FUNCTION_BLOCK E_CTU (* Event-Driven Up Counter *)
  (* Standard: 61499-1-A.18; Classification: Event-driven blocks; Function: Up-counter *)
  (* Version 0.1, 2001-04-27, JHC, Rockwell Automation, XML version *)
  (* Version 0.0, 1999-01-22, JHC, Rockwell Automation, SRC version *)
  (* Compiler header: package fb.rt.event; *)
  (* Compiler Java IBM VisualAge 3.0 *)
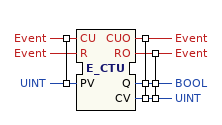
  EVENT_INPUT
    CU WITH PV; (* Count Up *)
    R; (* Reset *)
  END_EVENT
  EVENT_OUTPUT
    CUO WITH Q, CV; (* Count Up Output Event *)
    RO WITH Q, CV; (* Reset Output Event *)
  END_EVENT
  VAR_INPUT
    PV : UINT; (* Preset Value *)
  END_VAR
  VAR_OUTPUT
    Q : BOOL; (* CV==PV *)
    CV : UINT;
  END_VAR
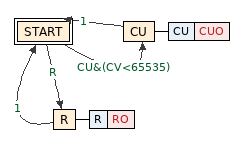
  EC_STATES
    START;
    CU : CU -> CUO;
    R : R -> RO;
  END_STATES
  EC_TRANSITIONS
    START TO CU := CU&(CV<65535);
    CU TO START := 1;
    START TO R := R;
    R TO START := 1;
  END_TRANSITIONS
  ALGORITHM CU IN ST: (* Count Up *)
CV:=CV+1;
Q:=(CV>=PV);
  END_ALGORITHM
  ALGORITHM R IN ST: (* Reset *)
CV:=0;
Q:=0;
  END_ALGORITHM
END_FUNCTION_BLOCK
